TYPE ST_ExtController_Set :
STRUCT
	b_available				: BOOL;
END_STRUCT
END_TYPE

(* stored: Version 1.1.0.1, ProductVersion 3.1.4026.18
   DUT ST_ExtController_Set: Id {9d99ae19-2b04-4caf-b3af-7cc0aa67da30} *)
